(* CoDeSys 2.3 export: FUZSIGNALTOVOLTAGEOUTPUT.EXP *)

(* POU K14/fUZSignalToVoltageOutput, ST *)
FUNCTION fUZSignalToVoltageOutput : REAL
(*
	Функция преобразования входного
	сигнала 0-100% в выходное управляющее
	напряжение на насос
*)
VAR_INPUT
	IN : USINT; (*Входной сигнал*)
END_VAR
VAR
END_VAR
(*TODO: написать корректную функцию преобразования тока в напряжение*)
fUZSignalToVoltageOutput := IN/10.0;
END_FUNCTION
